KUKA KRL program: check_ros_version.src, check_ros_version.dat

--- check_ros_version.src ---
&ACCESS RVP
&PARAM TEMPLATE = C:\KRC\Roboter\Template\vorgabe
&PARAM EDITMASK = *
DEF check_ros_version(major:IN, minor:IN, revision:IN)
  ; =============================================
  ; Copyright 2026 KUKA Hungaria Kft.
  ;
  ; Licensed under the Apache License, Version 2.0 (the "License");
  ; you may not use this file except in compliance with the License.
  ; You may obtain a copy of the License at
  ;
  ;     http://www.apache.org/licenses/LICENSE-2.0
  ;
  ; Unless required by applicable law or agreed to in writing, software
  ; distributed under the License is distributed on an "AS IS" BASIS,
  ; WITHOUT WARRANTIES OR CONDITIONS OF ANY KIND, either express or implied.
  ; See the License for the specific language governing permissions and
  ; limitations under the License.
  ; =============================================

  ; Compares the client-supplied semantic version against the rosruntime.dat globals
  DECL REAL major
  DECL REAL minor
  DECL REAL revision

  IF (major <> ROSRUNTIME_VERSION_MAJOR) OR (minor <> ROSRUNTIME_VERSION_MINOR) OR (revision <> ROSRUNTIME_VERSION_REV) THEN
    ; TODO: verify on the real controller which numeric ERRORID this HALT surfaces as
    ; on the C++ side (kRosRuntimeVersionMismatchErrorId in kss/mxa/client.h) and adjust it to match
    HALT
  ENDIF
END

--- check_ros_version.dat ---
&ACCESS R
DEFDAT check_ros_version PUBLIC
    GLOBAL REAL ROSRUNTIME_VERSION_MAJOR = 1.0
    GLOBAL REAL ROSRUNTIME_VERSION_MINOR = 0.0
    GLOBAL REAL ROSRUNTIME_VERSION_REV = 0.0
ENDDAT
